(* Logix 5000 project; controller cal1632 1756-L62 rev 16.20; software revision 16.05; part 25 of 61 *)
(* tags used below, declared in another part *)
   FAULT : BOOL;
   HMI : BOOL;
   p01_param_oven_timer_presets : DINT[32];
   p01_recipe_active : recipe;
   p01_sys_lc : Limit_Clamp;
   p01r09_pb_global_reset : BOOL;
   p02_dint_from_hmi : hmi_dint;
   p02_real_from_hmi : hmi_real;
   p19_ai_tc01 : REAL;
   p19_ao_cv : REAL;
   p19_di_tc01_bo : BOOL;
   p19_dint_to_hmi : DINT[16];
   p19_param_pid1_ff : REAL;
   p19_param_pid1_kd : REAL;
   p19_param_pid1_ki : REAL;
   p19_param_pid1_kp : REAL;
   p19_param_pid2_ff : REAL;
   p19_param_pid2_kd : REAL;
   p19_param_pid2_ki : REAL;
   p19_param_pid2_kp : REAL;
   p19_param_tc01_dev : REAL;
   p19_param_tc01z : REAL;
   p19_param_tc02z : REAL;
   p19_param_zone_pressure : REAL;
   p19r02_timer_warning : TIMER[4];
   p19r08 : routine;
   p19r08_timer_fault : TIMER[4];
   p19r08_timer_warning : TIMER[4];
   p19r09 : routine;
   p19r09_timer_fault : TIMER[4];
   p19r09_timer_warning : TIMER[4];
   p19r10 : routine;
   p19r10_timer_fault : TIMER[4];
   p19r10_timer_warning : TIMER[4];
   p19r16_pid_temp_cv : DINT;
   p19r30 : routine;
   p19r30_cv_man_sp : REAL;
   p19r30_pb_auto : BOOL;
   p19r30_pb_manual : BOOL;
   p19r30_pb_zone_off : BOOL;
   p19r30_pb_zone_on : BOOL;
   p19r30_permissive_run : BOOL;
   p19r30_pid_temp : PID;
   p19r30_pid_temp_pv : DINT;
   p19r30_pid_temp_sp : DINT;
   p19r30_request_cool : BOOL;
   p19r30_request_manual : BOOL;
   p19r30_timer_fault : TIMER[4];
   p19r30_timer_warning : TIMER[4];
   p19r31 : routine;
   p19r31_timer_fault : TIMER[4];
(* P19_Advanced_Cooling, continued *)

ROUTINE R08_Warnings   (* ladder *)
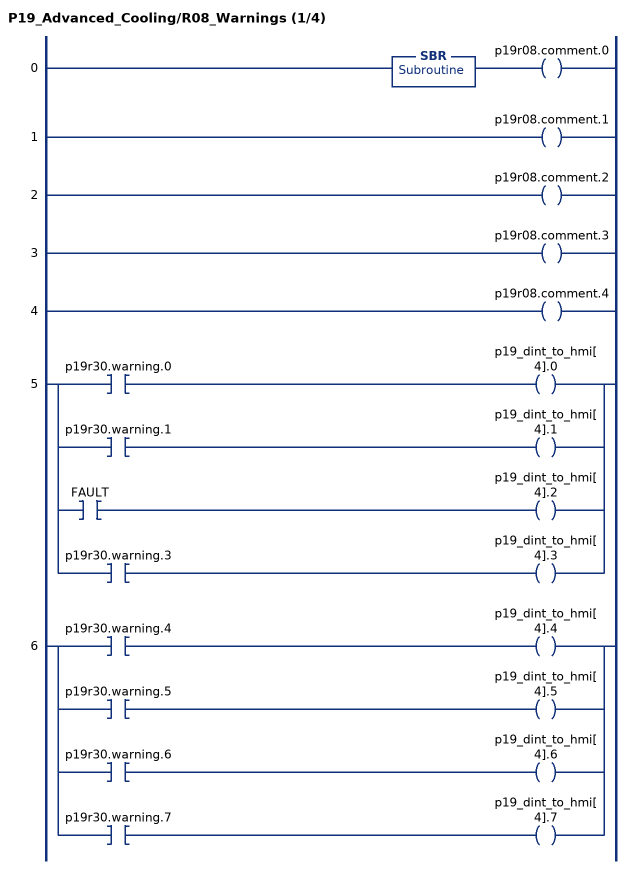
   0: SBR()OTE(p19r08.comment.0);
   1: OTE(p19r08.comment.1);
   2: OTE(p19r08.comment.2);
   3: OTE(p19r08.comment.3);
   4: OTE(p19r08.comment.4);
   5: [XIC(p19r30.warning.0) OTE(p19_dint_to_hmi[4].0) ,XIC(p19r30.warning.1) OTE(p19_dint_to_hmi[4].1) ,XIC(FAULT) OTE(p19_dint_to_hmi[4].2) ,XIC(p19r30.warning.3) OTE(p19_dint_to_hmi[4].3) ];
   6: [XIC(p19r30.warning.4) OTE(p19_dint_to_hmi[4].4) ,XIC(p19r30.warning.5) OTE(p19_dint_to_hmi[4].5) ,XIC(p19r30.warning.6) OTE(p19_dint_to_hmi[4].6) ,XIC(p19r30.warning.7) OTE(p19_dint_to_hmi[4].7) ];
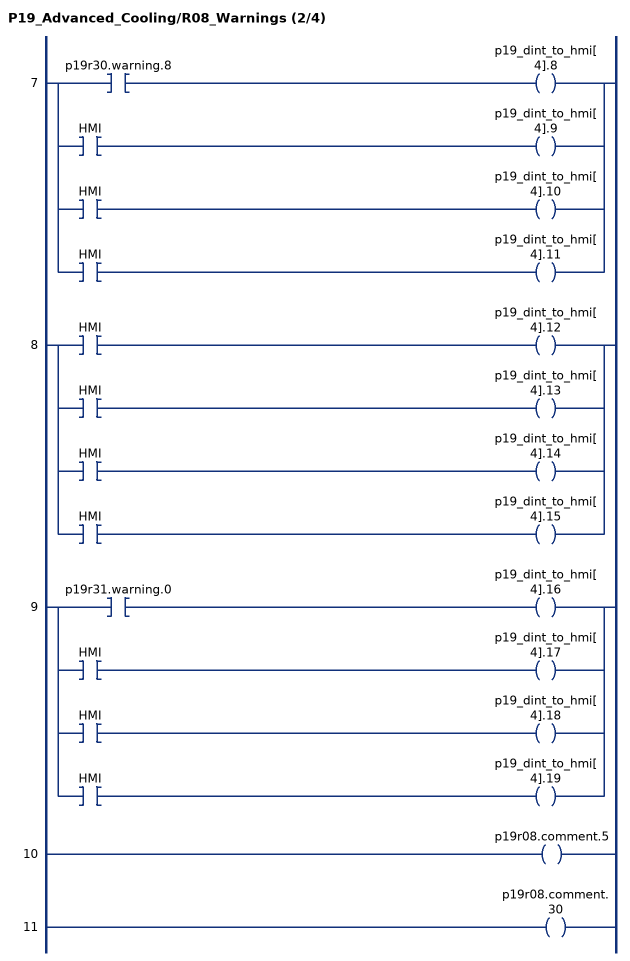
   7: [XIC(p19r30.warning.8) OTE(p19_dint_to_hmi[4].8) ,XIC(HMI) OTE(p19_dint_to_hmi[4].9) ,XIC(HMI) OTE(p19_dint_to_hmi[4].10) ,XIC(HMI) OTE(p19_dint_to_hmi[4].11) ];
   8: [XIC(HMI) OTE(p19_dint_to_hmi[4].12) ,XIC(HMI) OTE(p19_dint_to_hmi[4].13) ,XIC(HMI) OTE(p19_dint_to_hmi[4].14) ,XIC(HMI) OTE(p19_dint_to_hmi[4].15) ];
   9: [XIC(p19r31.warning.0) OTE(p19_dint_to_hmi[4].16) ,XIC(HMI) OTE(p19_dint_to_hmi[4].17) ,XIC(HMI) OTE(p19_dint_to_hmi[4].18) ,XIC(HMI) OTE(p19_dint_to_hmi[4].19) ];
   10: OTE(p19r08.comment.5);
   11: OTE(p19r08.comment.30);
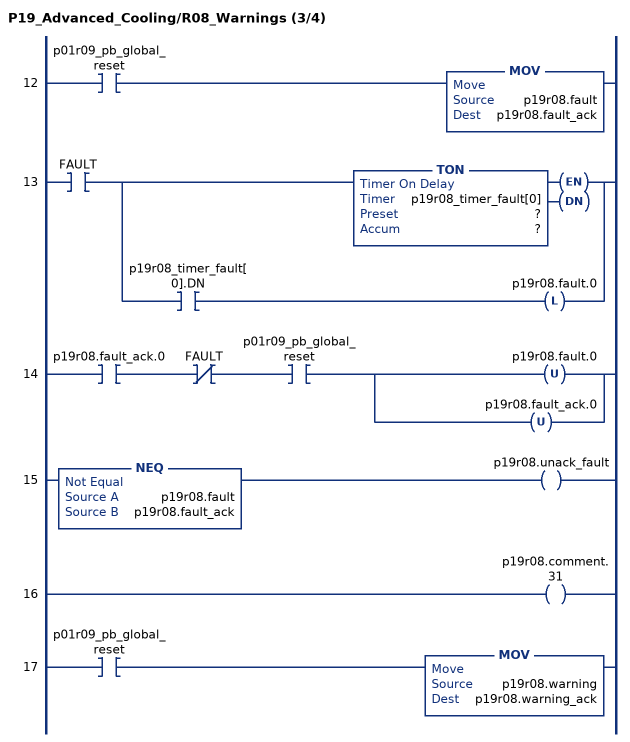
   12: XIC(p01r09_pb_global_reset)MOV(p19r08.fault,p19r08.fault_ack);
   13: XIC(FAULT)[TON(p19r08_timer_fault[0],?,?) ,XIC(p19r08_timer_fault[0].DN) OTL(p19r08.fault.0) ];
   14: XIC(p19r08.fault_ack.0)XIO(FAULT)XIC(p01r09_pb_global_reset)[OTU(p19r08.fault.0) ,OTU(p19r08.fault_ack.0) ];
   15: NEQ(p19r08.fault,p19r08.fault_ack)OTE(p19r08.unack_fault);
   16: OTE(p19r08.comment.31);
   17: XIC(p01r09_pb_global_reset)MOV(p19r08.warning,p19r08.warning_ack);
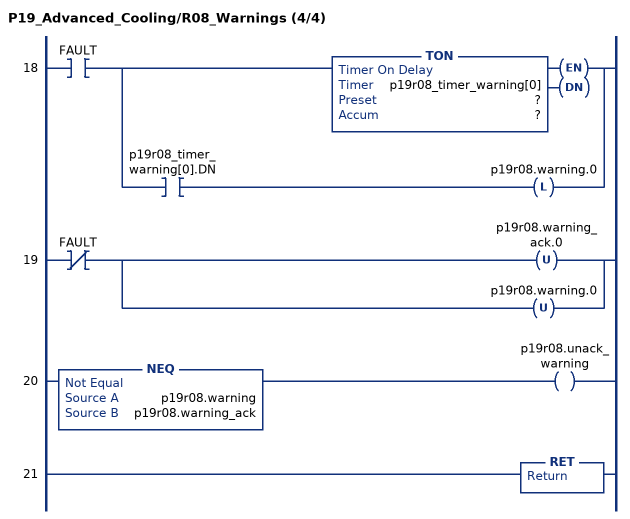
   18: XIC(FAULT)[TON(p19r08_timer_warning[0],?,?) ,XIC(p19r08_timer_warning[0].DN) OTL(p19r08.warning.0) ];
   19: XIO(FAULT)[OTU(p19r08.warning_ack.0) ,OTU(p19r08.warning.0) ];
   20: NEQ(p19r08.warning,p19r08.warning_ack)OTE(p19r08.unack_warning);
   21: RET();
END_ROUTINE

ROUTINE R09_Modes   (* ladder *)
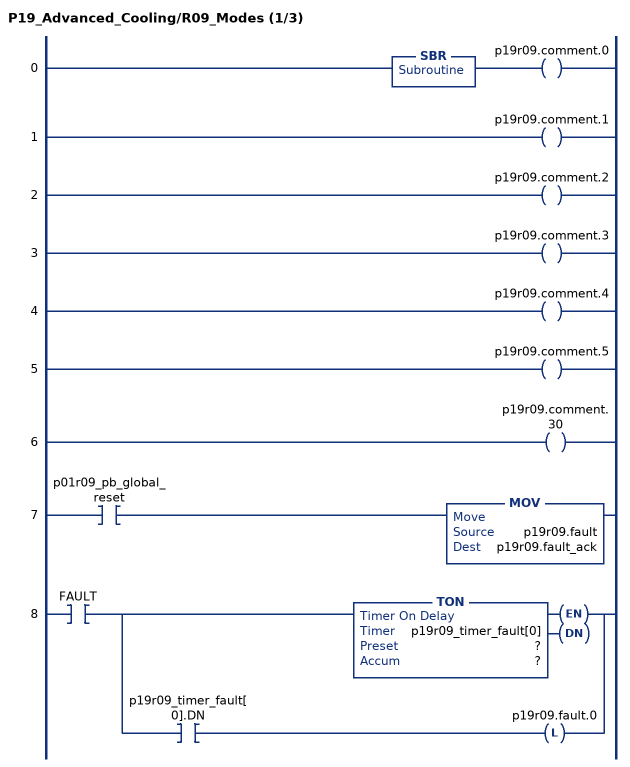
   0: SBR()OTE(p19r09.comment.0);
   1: OTE(p19r09.comment.1);
   2: OTE(p19r09.comment.2);
   3: OTE(p19r09.comment.3);
   4: OTE(p19r09.comment.4);
   5: OTE(p19r09.comment.5);
   6: OTE(p19r09.comment.30);
   7: XIC(p01r09_pb_global_reset)MOV(p19r09.fault,p19r09.fault_ack);
   8: XIC(FAULT)[TON(p19r09_timer_fault[0],?,?) ,XIC(p19r09_timer_fault[0].DN) OTL(p19r09.fault.0) ];
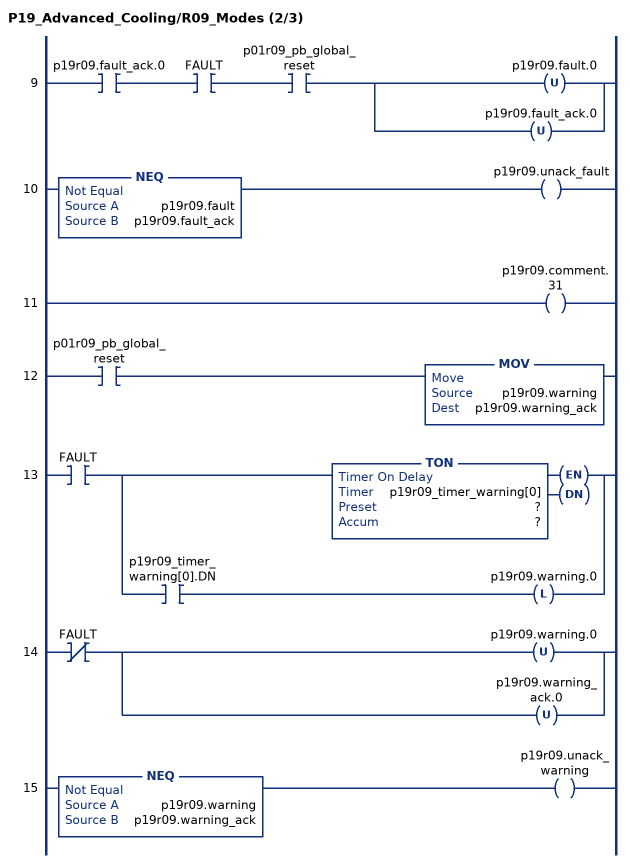
   9: XIC(p19r09.fault_ack.0)XIC(FAULT)XIC(p01r09_pb_global_reset)[OTU(p19r09.fault.0) ,OTU(p19r09.fault_ack.0) ];
   10: NEQ(p19r09.fault,p19r09.fault_ack)OTE(p19r09.unack_fault);
   11: OTE(p19r09.comment.31);
   12: XIC(p01r09_pb_global_reset)MOV(p19r09.warning,p19r09.warning_ack);
   13: XIC(FAULT)[TON(p19r09_timer_warning[0],?,?) ,XIC(p19r09_timer_warning[0].DN) OTL(p19r09.warning.0) ];
   14: XIO(FAULT)[OTU(p19r09.warning.0) ,OTU(p19r09.warning_ack.0) ];
   15: NEQ(p19r09.warning,p19r09.warning_ack)OTE(p19r09.unack_warning);
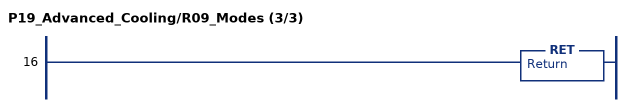
   16: RET();
END_ROUTINE

ROUTINE R10_Parameters   (* ladder *)
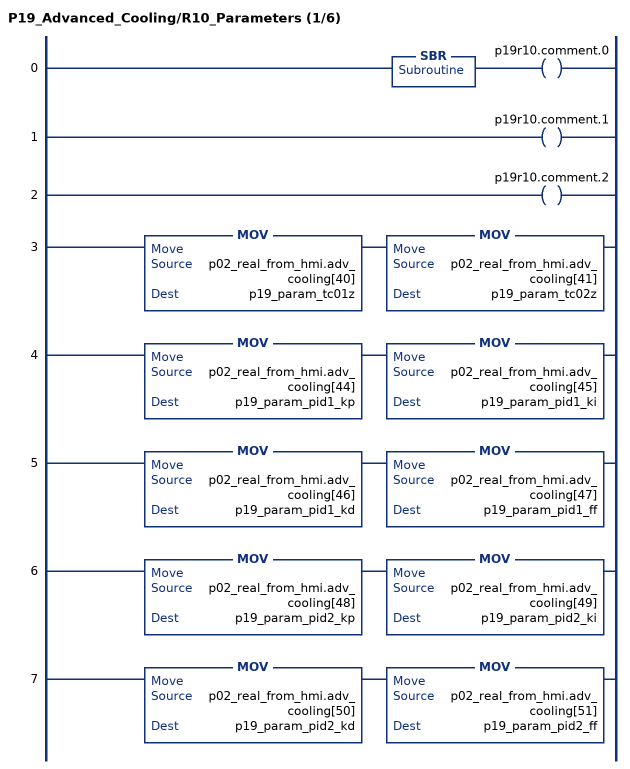
   0: SBR()OTE(p19r10.comment.0);
   1: OTE(p19r10.comment.1);
   2: OTE(p19r10.comment.2);
   3: MOV(p02_real_from_hmi.adv_cooling[40],p19_param_tc01z)MOV(p02_real_from_hmi.adv_cooling[41],p19_param_tc02z);
   4: MOV(p02_real_from_hmi.adv_cooling[44],p19_param_pid1_kp)MOV(p02_real_from_hmi.adv_cooling[45],p19_param_pid1_ki);
   5: MOV(p02_real_from_hmi.adv_cooling[46],p19_param_pid1_kd)MOV(p02_real_from_hmi.adv_cooling[47],p19_param_pid1_ff);
   6: MOV(p02_real_from_hmi.adv_cooling[48],p19_param_pid2_kp)MOV(p02_real_from_hmi.adv_cooling[49],p19_param_pid2_ki);
   7: MOV(p02_real_from_hmi.adv_cooling[50],p19_param_pid2_kd)MOV(p02_real_from_hmi.adv_cooling[51],p19_param_pid2_ff);
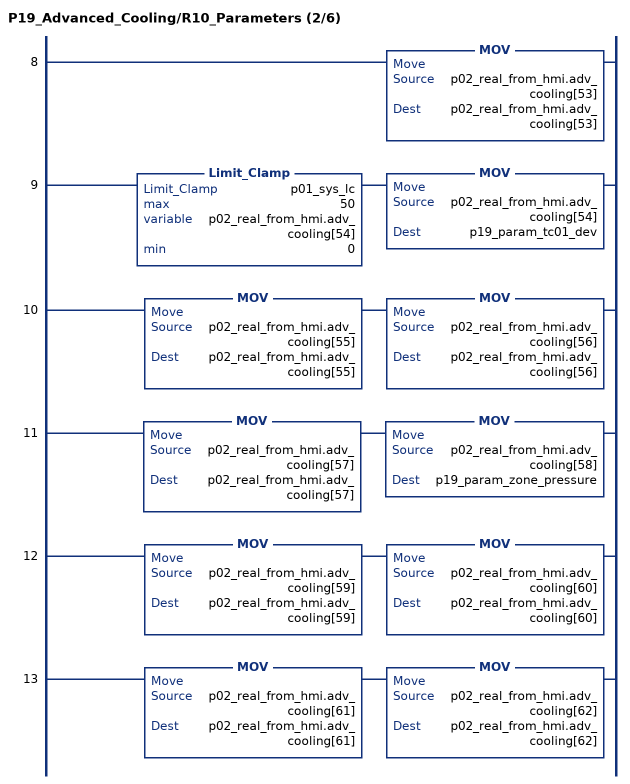
   8: MOV(p02_real_from_hmi.adv_cooling[53],p02_real_from_hmi.adv_cooling[53]);
   9: Limit_Clamp(p01_sys_lc,50,p02_real_from_hmi.adv_cooling[54],0)MOV(p02_real_from_hmi.adv_cooling[54],p19_param_tc01_dev);
   10: MOV(p02_real_from_hmi.adv_cooling[55],p02_real_from_hmi.adv_cooling[55])MOV(p02_real_from_hmi.adv_cooling[56],p02_real_from_hmi.adv_cooling[56]);
   11: MOV(p02_real_from_hmi.adv_cooling[57],p02_real_from_hmi.adv_cooling[57])MOV(p02_real_from_hmi.adv_cooling[58],p19_param_zone_pressure);
   12: MOV(p02_real_from_hmi.adv_cooling[59],p02_real_from_hmi.adv_cooling[59])MOV(p02_real_from_hmi.adv_cooling[60],p02_real_from_hmi.adv_cooling[60]);
   13: MOV(p02_real_from_hmi.adv_cooling[61],p02_real_from_hmi.adv_cooling[61])MOV(p02_real_from_hmi.adv_cooling[62],p02_real_from_hmi.adv_cooling[62]);
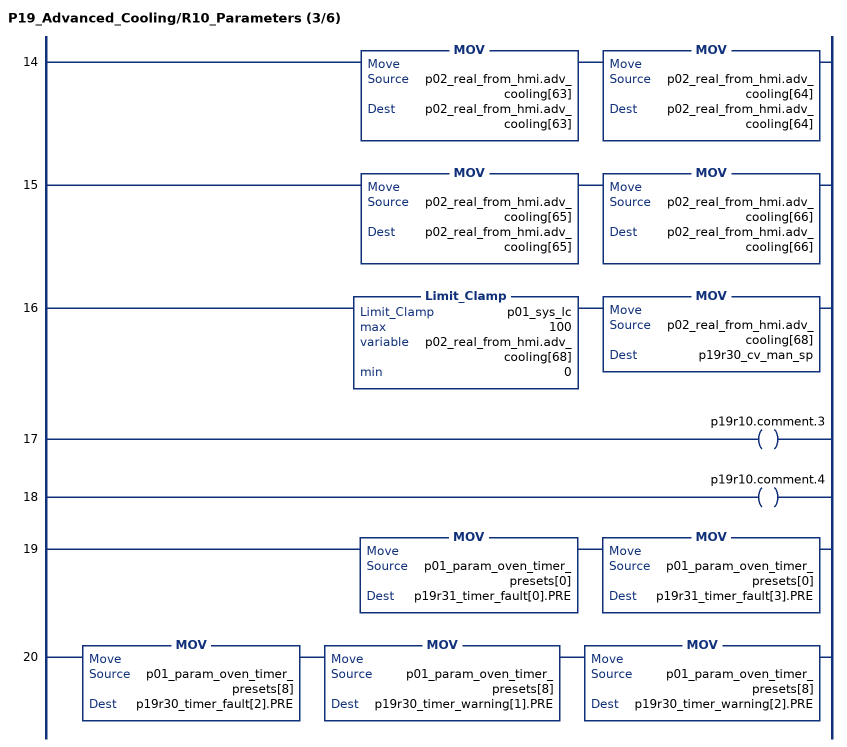
   14: MOV(p02_real_from_hmi.adv_cooling[63],p02_real_from_hmi.adv_cooling[63])MOV(p02_real_from_hmi.adv_cooling[64],p02_real_from_hmi.adv_cooling[64]);
   15: MOV(p02_real_from_hmi.adv_cooling[65],p02_real_from_hmi.adv_cooling[65])MOV(p02_real_from_hmi.adv_cooling[66],p02_real_from_hmi.adv_cooling[66]);
   16: Limit_Clamp(p01_sys_lc,100,p02_real_from_hmi.adv_cooling[68],0)MOV(p02_real_from_hmi.adv_cooling[68],p19r30_cv_man_sp);
   17: OTE(p19r10.comment.3);
   18: OTE(p19r10.comment.4);
   19: MOV(p01_param_oven_timer_presets[0],p19r31_timer_fault[0].PRE)MOV(p01_param_oven_timer_presets[0],p19r31_timer_fault[3].PRE);
   20: MOV(p01_param_oven_timer_presets[8],p19r30_timer_fault[2].PRE)MOV(p01_param_oven_timer_presets[8],p19r30_timer_warning[1].PRE)MOV(p01_param_oven_timer_presets[8],p19r30_timer_warning[2].PRE);
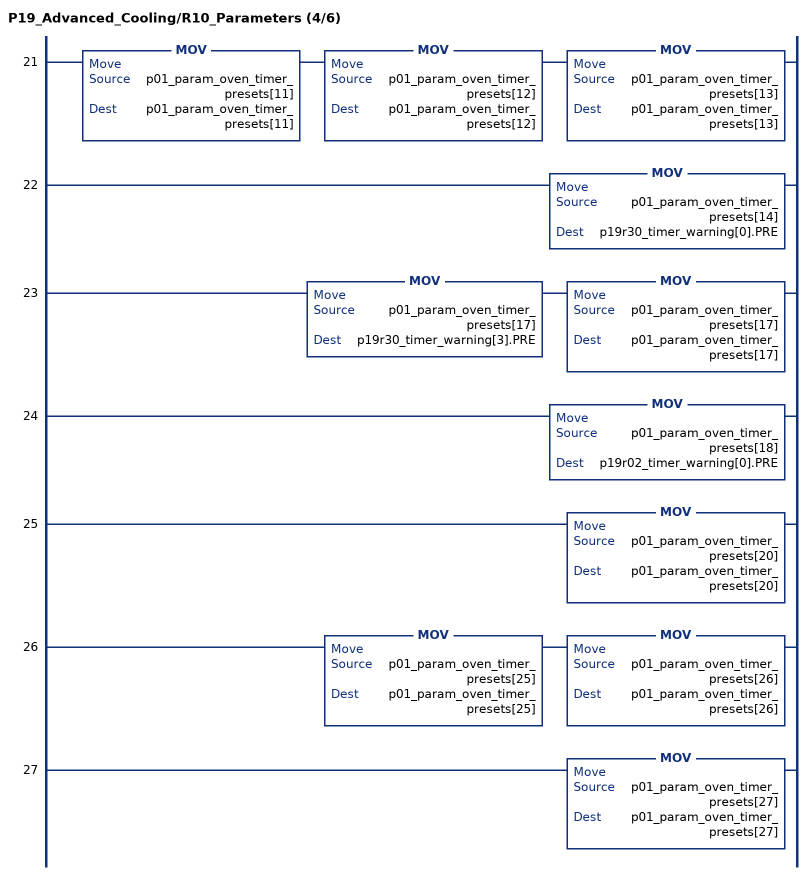
   21: MOV(p01_param_oven_timer_presets[11],p01_param_oven_timer_presets[11])MOV(p01_param_oven_timer_presets[12],p01_param_oven_timer_presets[12])MOV(p01_param_oven_timer_presets[13],p01_param_oven_timer_presets[13]);
   22: MOV(p01_param_oven_timer_presets[14],p19r30_timer_warning[0].PRE);
   23: MOV(p01_param_oven_timer_presets[17],p19r30_timer_warning[3].PRE)MOV(p01_param_oven_timer_presets[17],p01_param_oven_timer_presets[17]);
   24: MOV(p01_param_oven_timer_presets[18],p19r02_timer_warning[0].PRE);
   25: MOV(p01_param_oven_timer_presets[20],p01_param_oven_timer_presets[20]);
   26: MOV(p01_param_oven_timer_presets[25],p01_param_oven_timer_presets[25])MOV(p01_param_oven_timer_presets[26],p01_param_oven_timer_presets[26]);
   27: MOV(p01_param_oven_timer_presets[27],p01_param_oven_timer_presets[27]);
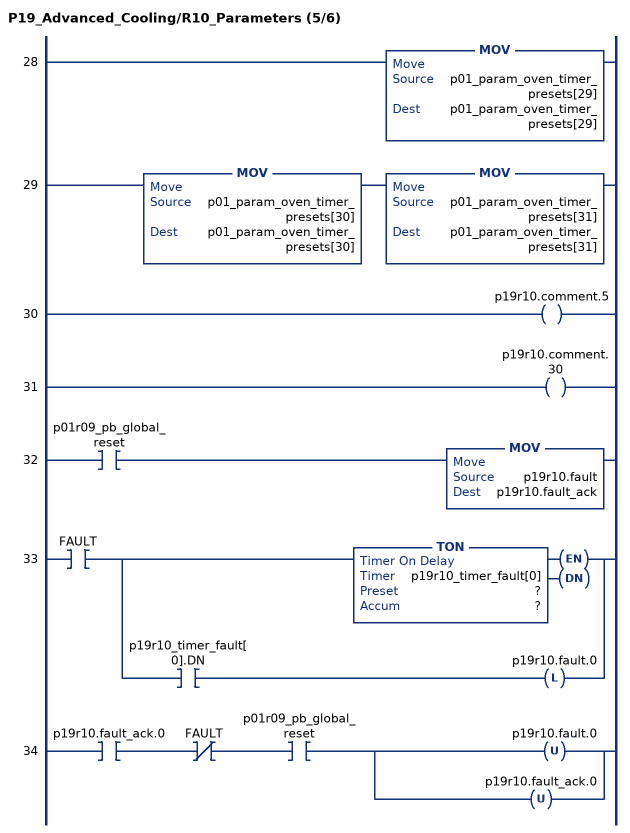
   28: MOV(p01_param_oven_timer_presets[29],p01_param_oven_timer_presets[29]);
   29: MOV(p01_param_oven_timer_presets[30],p01_param_oven_timer_presets[30])MOV(p01_param_oven_timer_presets[31],p01_param_oven_timer_presets[31]);
   30: OTE(p19r10.comment.5);
   31: OTE(p19r10.comment.30);
   32: XIC(p01r09_pb_global_reset)MOV(p19r10.fault,p19r10.fault_ack);
   33: XIC(FAULT)[TON(p19r10_timer_fault[0],?,?) ,XIC(p19r10_timer_fault[0].DN) OTL(p19r10.fault.0) ];
   34: XIC(p19r10.fault_ack.0)XIO(FAULT)XIC(p01r09_pb_global_reset)[OTU(p19r10.fault.0) ,OTU(p19r10.fault_ack.0) ];
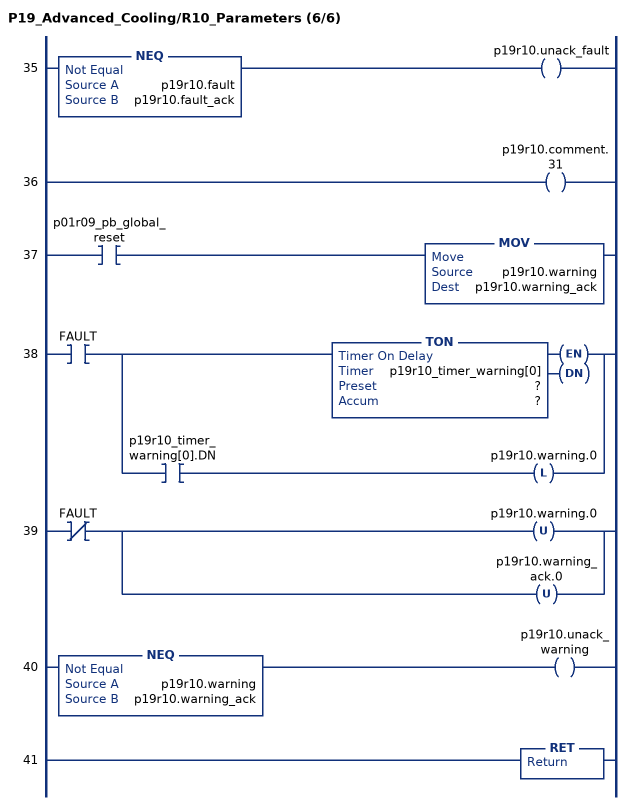
   35: NEQ(p19r10.fault,p19r10.fault_ack)OTE(p19r10.unack_fault);
   36: OTE(p19r10.comment.31);
   37: XIC(p01r09_pb_global_reset)MOV(p19r10.warning,p19r10.warning_ack);
   38: XIC(FAULT)[TON(p19r10_timer_warning[0],?,?) ,XIC(p19r10_timer_warning[0].DN) OTL(p19r10.warning.0) ];
   39: XIO(FAULT)[OTU(p19r10.warning.0) ,OTU(p19r10.warning_ack.0) ];
   40: NEQ(p19r10.warning,p19r10.warning_ack)OTE(p19r10.unack_warning);
   41: RET();
END_ROUTINE

ROUTINE R30_Temperature_Control   (* ladder *)
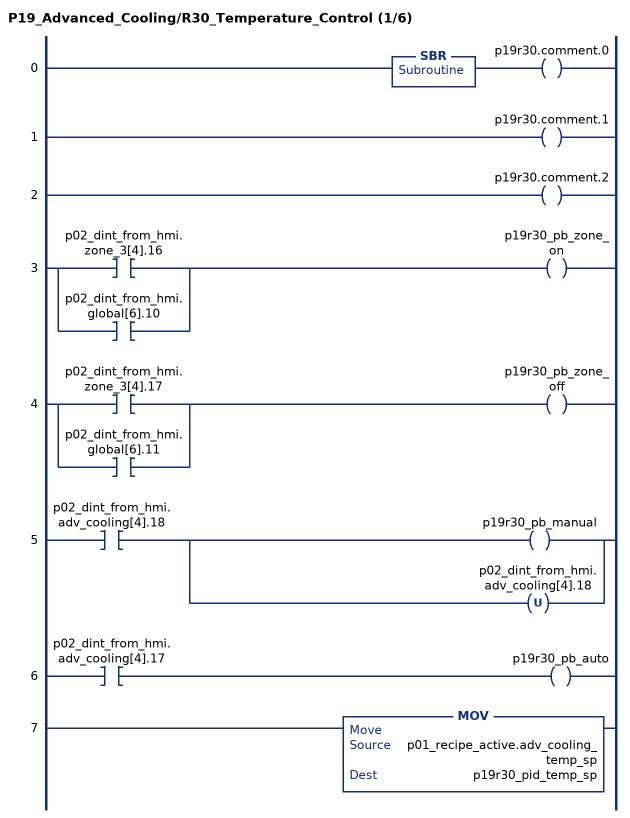
   0: SBR()OTE(p19r30.comment.0);
   1: OTE(p19r30.comment.1);
   2: OTE(p19r30.comment.2);
   3: [XIC(p02_dint_from_hmi.zone_3[4].16) ,XIC(p02_dint_from_hmi.global[6].10) ]OTE(p19r30_pb_zone_on);
   4: [XIC(p02_dint_from_hmi.zone_3[4].17) ,XIC(p02_dint_from_hmi.global[6].11) ]OTE(p19r30_pb_zone_off);
   5: XIC(p02_dint_from_hmi.adv_cooling[4].18)[OTE(p19r30_pb_manual) ,OTU(p02_dint_from_hmi.adv_cooling[4].18) ];
   6: XIC(p02_dint_from_hmi.adv_cooling[4].17)OTE(p19r30_pb_auto);
   7: MOV(p01_recipe_active.adv_cooling_temp_sp,p19r30_pid_temp_sp);
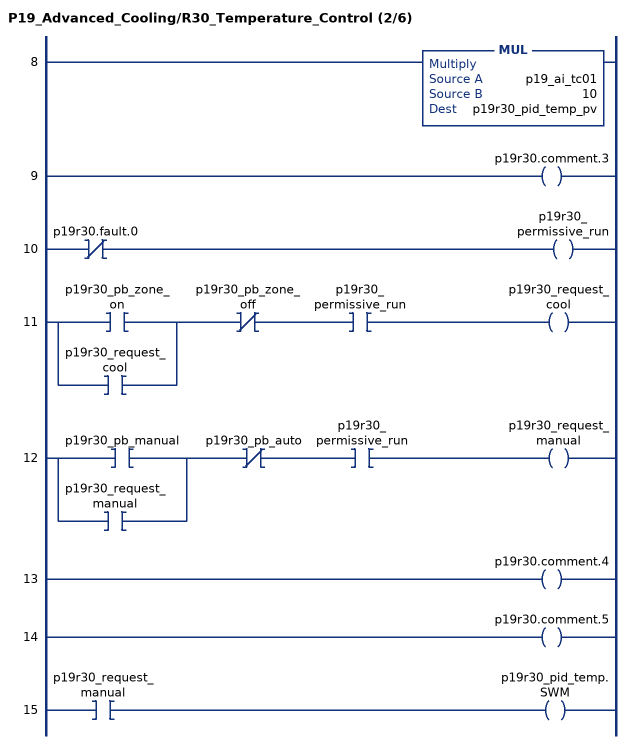
   8: MUL(p19_ai_tc01,10,p19r30_pid_temp_pv);
   9: OTE(p19r30.comment.3);
   10: XIO(p19r30.fault.0)OTE(p19r30_permissive_run);
   11: [XIC(p19r30_pb_zone_on) ,XIC(p19r30_request_cool) ]XIO(p19r30_pb_zone_off)XIC(p19r30_permissive_run)OTE(p19r30_request_cool);
   12: [XIC(p19r30_pb_manual) ,XIC(p19r30_request_manual) ]XIO(p19r30_pb_auto)XIC(p19r30_permissive_run)OTE(p19r30_request_manual);
   13: OTE(p19r30.comment.4);
   14: OTE(p19r30.comment.5);
   15: XIC(p19r30_request_manual)OTE(p19r30_pid_temp.SWM);
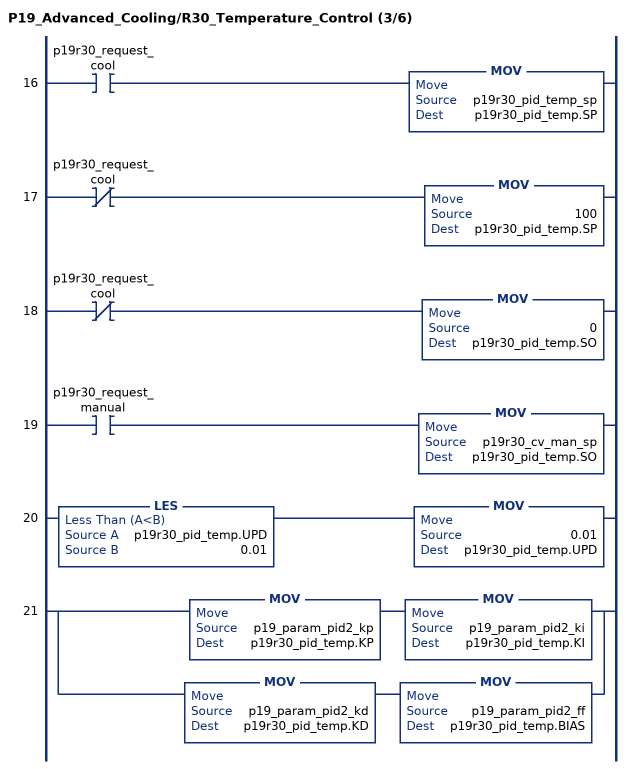
   16: XIC(p19r30_request_cool)MOV(p19r30_pid_temp_sp,p19r30_pid_temp.SP);
   17: XIO(p19r30_request_cool)MOV(100,p19r30_pid_temp.SP);
   18: XIO(p19r30_request_cool)MOV(0,p19r30_pid_temp.SO);
   19: XIC(p19r30_request_manual)MOV(p19r30_cv_man_sp,p19r30_pid_temp.SO);
   20: LES(p19r30_pid_temp.UPD,0.01)MOV(0.01,p19r30_pid_temp.UPD);
   21: [MOV(p19_param_pid2_kp,p19r30_pid_temp.KP) MOV(p19_param_pid2_ki,p19r30_pid_temp.KI) ,MOV(p19_param_pid2_kd,p19r30_pid_temp.KD) MOV(p19_param_pid2_ff,p19r30_pid_temp.BIAS) ];
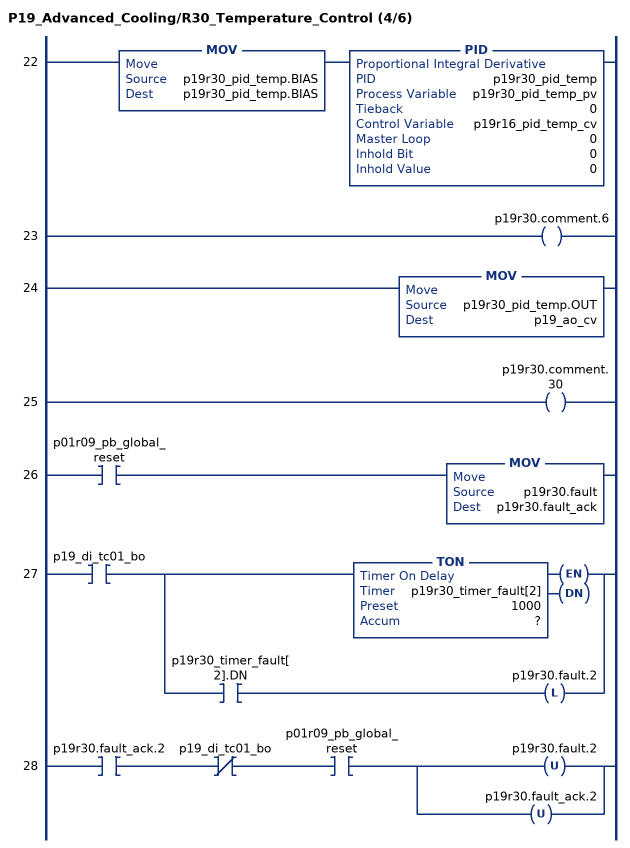
   22: MOV(p19r30_pid_temp.BIAS,p19r30_pid_temp.BIAS)PID(p19r30_pid_temp,p19r30_pid_temp_pv,0,p19r16_pid_temp_cv,0,0,0);
   23: OTE(p19r30.comment.6);
   24: MOV(p19r30_pid_temp.OUT,p19_ao_cv);
   25: OTE(p19r30.comment.30);
   26: XIC(p01r09_pb_global_reset)MOV(p19r30.fault,p19r30.fault_ack);
   27: XIC(p19_di_tc01_bo)[TON(p19r30_timer_fault[2],?,?) ,XIC(p19r30_timer_fault[2].DN) OTL(p19r30.fault.2) ];
   28: XIC(p19r30.fault_ack.2)XIO(p19_di_tc01_bo)XIC(p01r09_pb_global_reset)[OTU(p19r30.fault.2) ,OTU(p19r30.fault_ack.2) ];
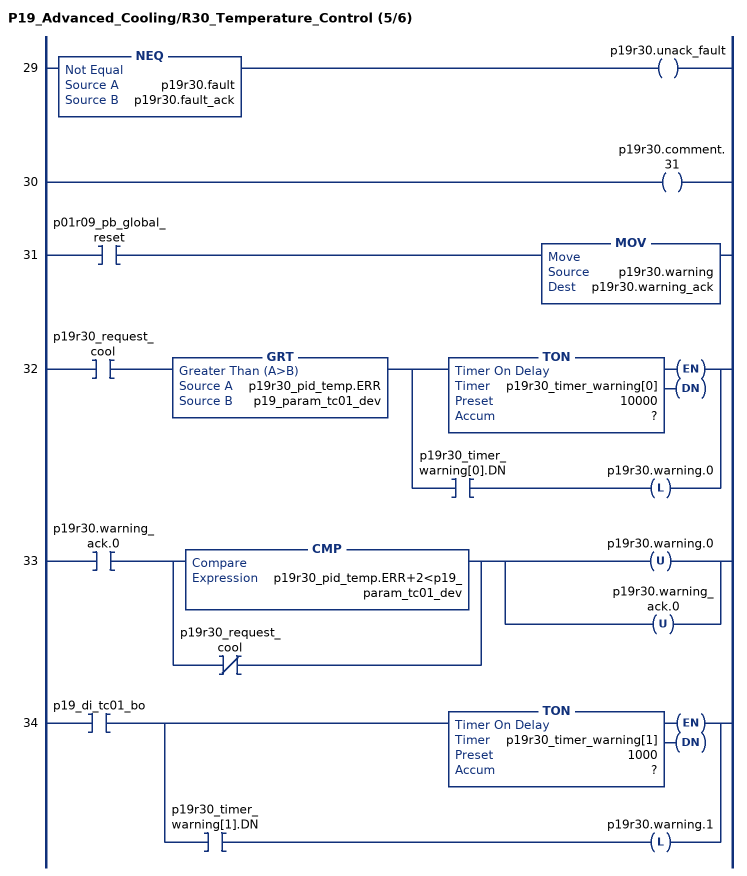
   29: NEQ(p19r30.fault,p19r30.fault_ack)OTE(p19r30.unack_fault);
   30: OTE(p19r30.comment.31);
   31: XIC(p01r09_pb_global_reset)MOV(p19r30.warning,p19r30.warning_ack);
   32: XIC(p19r30_request_cool)GRT(p19r30_pid_temp.ERR,p19_param_tc01_dev)[TON(p19r30_timer_warning[0],?,?) ,XIC(p19r30_timer_warning[0].DN) OTL(p19r30.warning.0) ];
   33: XIC(p19r30.warning_ack.0)[CMP(p19r30_pid_temp.ERR+2<p19_param_tc01_dev) ,XIO(p19r30_request_cool) ][OTU(p19r30.warning.0) ,OTU(p19r30.warning_ack.0) ];
   34: XIC(p19_di_tc01_bo)[TON(p19r30_timer_warning[1],?,?) ,XIC(p19r30_timer_warning[1].DN) OTL(p19r30.warning.1) ];
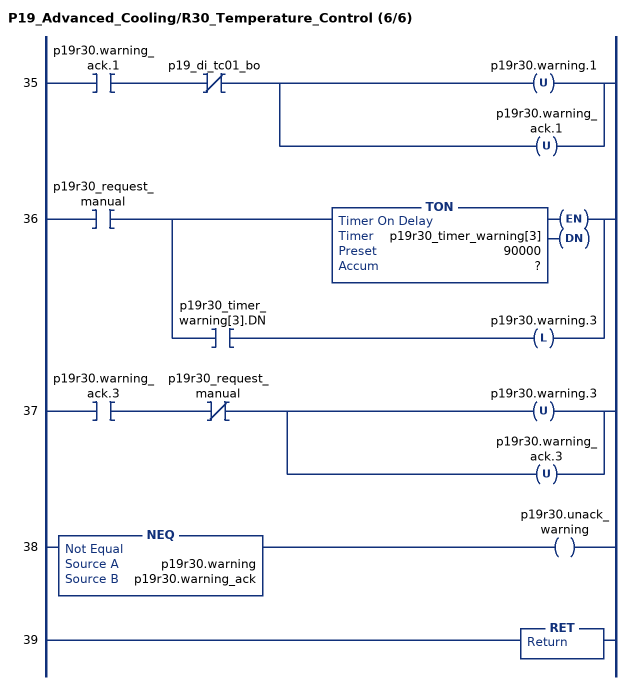
   35: XIC(p19r30.warning_ack.1)XIO(p19_di_tc01_bo)[OTU(p19r30.warning.1) ,OTU(p19r30.warning_ack.1) ];
   36: XIC(p19r30_request_manual)[TON(p19r30_timer_warning[3],?,?) ,XIC(p19r30_timer_warning[3].DN) OTL(p19r30.warning.3) ];
   37: XIC(p19r30.warning_ack.3)XIO(p19r30_request_manual)[OTU(p19r30.warning.3) ,OTU(p19r30.warning_ack.3) ];
   38: NEQ(p19r30.warning,p19r30.warning_ack)OTE(p19r30.unack_warning);
   39: RET();
END_ROUTINE
